TYPE
    DUT_IncomingMsgRequest :
    STRUCT
        reqHdr : DUT_MsgToAmsPortHeader;
        reqData : ARRAY[0..991] OF BYTE;
    END_STRUCT
END_TYPE

(* stored: Version 1.1.0.1, ProductVersion 3.1.4024.12
   DUT DUT_IncomingMsgRequest: Id {7b021bd8-da94-4954-8897-62c19ed6a9ed} *)
